(* IEC 61131-3 sources: plcassist-cli/packages/volt-lsp-iec/test-corpus/pro2193/Device/Plc Logic/Application/02 Processes/21 SER/2120 - Transfer Control/Products, 8 files *)

(* ---- TransferProducts_ChainToReject_WithCarrierPlatesFB.fb ---- *)
{attribute 'symbol' := 'none'}
{attribute 'monitoring_display' := 'ActState'}
FUNCTION_BLOCK TransferProducts_ChainToReject_WithCarrierPlatesFB
EXTENDS Transfer_BaseFB
IMPLEMENTS IModuleTransferExecute
VAR_INPUT
	chain					: IChain_WithCarrierPlates_TransferOuttake_Commands;
	reject					: IRejectStation_Base_Commands;
END_VAR
VAR
	gettingProduct			: ARRAY[1..GVL_Constants.ChainProductsForReject] OF BOOL;

	ActState :
	(
		StateNone							:= 0,
		StateRejectMovesInPosition			:= 100,
		StateRejectGetsProducts				:= 200,
		StateOpenProductCarriers			:= 250,
		StateCopyProductData				:= 300,
		StateFreeReject						:= 400,
		StateFinal							:= 999
	) DINT;

END_VAR

SUPER^();

// Enable manual control of Reject cylinders when chain is in safe position.
reject.ExternalManualControlEnabled := chain.InExactPosition();

END_FUNCTION_BLOCK

METHOD PUBLIC CheckIfTransferIsNeeded : BOOL
VAR_INPUT
	iParameter			: INT := 1;	// 0: Invalid, 1: Takeover Pos 1, etc.
END_VAR
VAR_INST
	product				: REFERENCE TO ProductType;
	i, j				: USINT;
END_VAR
// Go from first Reject vacuum, to the last.
FOR i := 1 TO GVL_Constants.ChainProductsForReject DO

	gettingProduct[i]		:= FALSE;

	// Copy reference to products from the chain
	product REF= chain.ReturnProduct(PersistentVars.RecipeVars.chainPos_Reject[i]);

	IF NOT __ISVALIDREF(product) THEN
		CONTINUE;
	END_IF

	FOR j := 1 TO GVL_Constants.MaxRejectReasonsTotal DO
		gettingProduct[i]	S= product.RejectReason[j] AND NOT product.RejectReasonIgnored[j];
	END_FOR

	gettingProduct[i]		S= product.UncountedReject;
	gettingProduct[i]		S= product.SampleShot;

	// When reject is after z unit, always reject all products
	IF NOT gettingProduct[i] AND NOT chain.ZUnitIsAfterReject THEN
		product.UncountedReject	:= TRUE;
		gettingProduct[i]	:= TRUE;
	END_IF

	CheckIfTransferIsNeeded	S= gettingProduct[i];
END_FOR
END_METHOD

METHOD PROTECTED Cyclic
State(actState	:= ActState);
END_METHOD

// Command to reset the module (Statemachine to zero state) in case of E-Stop
METHOD PUBLIC EStop : BOOL	// Returns true when drives are in standstill
CommandLock.ForceRelease();

ActState	:= StateNone;
EStop		:= TRUE;
END_METHOD

// Start transfer of products or labels between 2 units
METHOD PUBLIC ExecuteTransfer : BOOL
VAR_INPUT
	iParameter : INT := 1;	// 0: Invalid, 1: Takeover Pos 1, etc.
END_VAR
IF NOT CommandLock.Request(__POUNAME()) THEN
	RETURN;
END_IF

IF CommandLock.FirstCall THEN
	;
END_IF

takeoverPosition := iParameter;	// Copy parameters

IF ActState = StateNone THEN
	ActState := StateRejectMovesInPosition;
END_IF

IF ActState = StateFinal THEN
	ExecuteTransfer := CommandLock.Release(__POUNAME());
END_IF
END_METHOD

METHOD PROTECTED Execute_Sequence1
VAR_INST
	data				: WORD;
	product				: REFERENCE TO ProductType;
	result				: ARRAY[1..2] OF BOOL;
END_VAR
VAR
	i					: USINT;
END_VAR
CASE ActState OF
	StateNone:
		;

	StateRejectMovesInPosition:
		IF chain.InPosition(10.0) THEN
			ActState := StateRejectGetsProducts;
		END_IF

	StateRejectGetsProducts:

		IF State.Changed THEN
			Arrays.Bool_Reset(result);
			data := 0;
			FOR i := 1 TO GVL_Constants.ChainProductsForReject DO
				BitLogic.Load(data, gettingProduct[i], i);	// set a bit number when we transfer a product.
			END_FOR
		END_IF

		result[1]	:= result[1] OR_ELSE reject.GetProducts(data);

		IF chain.InExactPosition() THEN
			ActState := StateOpenProductCarriers;
		END_IF

	StateOpenProductCarriers:
		result[1]	:= result[1] OR_ELSE reject.GetProducts(data);
		result[2]	:= result[2] OR_ELSE chain.RejectOpenProductCarriers();

		IF Arrays.Bool_All(result, TRUE) THEN
			ActState := StateCopyProductData;
		END_IF

	StateCopyProductData:
		FOR i := 1 TO GVL_Constants.ChainProductsForReject DO

			IF NOT gettingProduct[i] THEN
				CONTINUE;
			END_IF

			// Copy reference to products from the chain
			product REF= chain.ReturnProduct(PersistentVars.RecipeVars.chainPos_Reject[i]);

			// Reject is not able to fail to transfer the product (like the Z Unit)
			reject.CopyProductStatus(i, product);
			chain.ClearProductCarrier(PersistentVars.RecipeVars.chainPos_Reject[i]);
			gettingProduct[i] := FALSE;

		END_FOR

		ActState := StateFreeReject;

	StateFreeReject:
		IF State.Changed THEN
			Arrays.Bool_Reset(result);
		END_IF

		// The last step of the product transfer must always be: TransferComplete()
		// This lets the Z Unit know that the transfer is done.
		// The Z Unit decides if it moves to the next Takeover position, or stack the products.
		result[1]	:= result[1] OR_ELSE reject.TransferComplete();
		result[2]	:= result[2] OR_ELSE chain.RejectCloseProductCarriers();

		IF Arrays.Bool_All(result, TRUE) THEN
			ActState := StateFinal;
		END_IF

	StateFinal:
		ActState := StateNone;
END_CASE
END_METHOD

// Command to stop a module (Statemachine to zero state)
METHOD PUBLIC Stop : BOOL	// Returns true when drives are in standstill
CommandLock.ForceRelease();

ActState	:= StateNone;
Stop		:= TRUE;
END_METHOD

// Transfer has started and is doing something
{attribute 'monitoring':='call'}
PROPERTY TransferBusy : BOOL
GET
VAR
END_VAR
TransferBusy	:= ActState <> StateNone;
END_GET
END_PROPERTY

(* ---- TransferProducts_ChainToRejectFB.fb ---- *)
{attribute 'symbol' := 'none'}
{attribute 'monitoring_display' := 'ActState'}
FUNCTION_BLOCK TransferProducts_ChainToRejectFB
EXTENDS Transfer_BaseFB
IMPLEMENTS IModuleTransferExecute
VAR_INPUT
	chain					: IChain_Base_TransferOuttake_Commands;
	reject					: IRejectStation_Base_Commands;
END_VAR
VAR
	gettingProduct			: ARRAY[1..GVL_Constants.ChainProductsForReject] OF BOOL;

	ActState :
	(
		StateNone							:= 0,
		StateRejectMovesInPosition			:= 100,
		StateRejectGetsProducts				:= 200,
		StateCopyProductData				:= 300,
		StateFreeReject						:= 400,
		StateFinal							:= 999
	) DINT;

END_VAR

SUPER^();

// Enable manual control of Reject cylinders when chain is in safe position.
reject.ExternalManualControlEnabled := chain.InExactPosition();

END_FUNCTION_BLOCK

METHOD PUBLIC CheckIfTransferIsNeeded : BOOL
VAR_INPUT
	iParameter			: INT := 1;	// 0: Invalid, 1: Takeover Pos 1, etc.
END_VAR
VAR_INST
	product				: REFERENCE TO ProductType;
	i, j				: USINT;
END_VAR
// Go from first Reject vacuum, to the last.
FOR i := 1 TO GVL_Constants.ChainProductsForReject DO

	gettingProduct[i]		:= FALSE;

	// Copy reference to products from the chain
	product REF= chain.ReturnProduct(PersistentVars.RecipeVars.chainPos_Reject[i]);

	IF NOT __ISVALIDREF(product) THEN
		EXIT;
	END_IF

	gettingProduct[i]		:= FALSE;

	FOR j := 1 TO GVL_Constants.MaxRejectReasonsTotal DO
		gettingProduct[i]	S= product.RejectReason[j] AND NOT product.RejectReasonIgnored[j];
	END_FOR

	gettingProduct[i]		S= product.UncountedReject;
	gettingProduct[i]		S= product.SampleShot;

	CheckIfTransferIsNeeded	S= gettingProduct[i];

	IF NOT gettingProduct[i] THEN
		EXIT;
	END_IF

END_FOR
END_METHOD

METHOD PROTECTED Cyclic
State(actState	:= ActState);
END_METHOD

// Command to reset the module (Statemachine to zero state) in case of E-Stop
METHOD PUBLIC EStop : BOOL	// Returns true when drives are in standstill
CommandLock.ForceRelease();

ActState	:= StateNone;
EStop		:= TRUE;
END_METHOD

// Start transfer of products or labels between 2 units
METHOD PUBLIC ExecuteTransfer : BOOL
VAR_INPUT
	iParameter : INT := 1;	// 0: Invalid, 1: Takeover Pos 1, etc.
END_VAR
IF NOT CommandLock.Request(__POUNAME()) THEN
	RETURN;
END_IF

IF CommandLock.FirstCall THEN
	;
END_IF

takeoverPosition := iParameter;	// Copy parameters

IF ActState = StateNone THEN
	ActState := StateRejectMovesInPosition;
END_IF

IF ActState = StateFinal THEN
	ExecuteTransfer := CommandLock.Release(__POUNAME());
END_IF
END_METHOD

METHOD PROTECTED Execute_Sequence1
VAR_INST
	data				: WORD;
	product				: REFERENCE TO ProductType;
	result				: ARRAY[1..2] OF BOOL;
END_VAR
VAR
	i					: USINT;
END_VAR
CASE ActState OF
	StateNone:
		;

	StateRejectMovesInPosition:
		IF chain.InExactPosition() THEN
			ActState := StateRejectGetsProducts;
		END_IF

	StateRejectGetsProducts:
		IF State.Changed THEN
			Arrays.Bool_Reset(result);
			data := 0;
			FOR i := 1 TO GVL_Constants.ChainProductsForReject DO
				BitLogic.Load(data, gettingProduct[i], i);	// set a bit number when we transfer a product.
			END_FOR
		END_IF

		result[1]	:= result[1] OR_ELSE reject.GetProducts(data);
		result[2]	:= TRUE;

		IF Arrays.Bool_All(result, TRUE) THEN
			ActState := StateCopyProductData;
		END_IF

	StateCopyProductData:
		FOR i := 1 TO GVL_Constants.ChainProductsForReject DO

			IF NOT gettingProduct[i] THEN
				CONTINUE;
			END_IF

			// Copy reference to products from the chain
			product REF= chain.ReturnProduct(PersistentVars.RecipeVars.chainPos_Reject[i]);

			// Reject is not able to fail to transfer the product (like the Z Unit)
			reject.CopyProductStatus(i, product);
			chain.ClearProductCarrier(PersistentVars.RecipeVars.chainPos_Reject[i]);
			gettingProduct[i] := FALSE;

		END_FOR

		ActState := StateFreeReject;

	StateFreeReject:
		IF State.Changed THEN
			Arrays.Bool_Reset(result);
		END_IF

		// The last step of the product transfer must always be: TransferComplete()
		// This lets the Z Unit know that the transfer is done.
		// The Z Unit decides if it moves to the next Takeover position, or stack the products.
		result[1]	:= result[1] OR_ELSE reject.TransferComplete();
		result[2]	:= TRUE;

		IF Arrays.Bool_All(result, TRUE) THEN
			ActState := StateFinal;
		END_IF

	StateFinal:
		ActState := StateNone;
END_CASE
END_METHOD

// Command to stop a module (Statemachine to zero state)
METHOD PUBLIC Stop : BOOL	// Returns true when drives are in standstill
CommandLock.ForceRelease();

ActState	:= StateNone;
Stop		:= TRUE;
END_METHOD

// Transfer has started and is doing something
{attribute 'monitoring':='call'}
PROPERTY TransferBusy : BOOL
GET
VAR
END_VAR
TransferBusy	:= ActState <> StateNone;
END_GET
END_PROPERTY

(* ---- TransferProducts_ChainToZ_WithCarrierPlatesFB.fb ---- *)
{attribute 'symbol' := 'none'}
{attribute 'monitoring_display' := 'ActState'}
FUNCTION_BLOCK TransferProducts_ChainToZ_WithCarrierPlatesFB
EXTENDS Transfer_BaseFB
IMPLEMENTS IModuleTransferExecute
VAR_INPUT
	chain					: IChain_WithCarrierPlates_TransferOuttake_Commands;
	zUnit					: IZUnit_ForChainWithServoRotate_Transfer_Commands;
END_VAR
VAR
	result					: ARRAY[1..2] OF BOOL;
	gettingProduct			: ARRAY[1..GVL_Constants.ChainProductsForZUnit] OF BOOL;

	ActState :
	(
		StateNone							:= 0,
		StateZUnitMovesInPosition			:= 100,
		StateZUnitGetsProducts				:= 200,
		StateZUnitOpenProductCarriers		:= 300,
		StateZUnitRetractWithProducts		:= 400,
		StateCopyProductData				:= 500,
		StateFreeZUnit						:= 600,
		StateFinal							:= 999
	) DINT;

END_VAR

SUPER^();

// Enable manual control of Z Unit motor when chain is in safe position.
zUnit.ExternalManualControlEnabled := TRUE; //chain.InExactPosition();

END_FUNCTION_BLOCK

METHOD PUBLIC CheckIfTransferIsNeeded : BOOL
VAR_INPUT
	iParameter			: INT := 1;	// 0: Invalid, 1: Takeover Pos 1, etc.
END_VAR
VAR_INST
	product				: REFERENCE TO ProductType;
	zUnitGripperFilled	: BOOL;
	data				: WORD;
END_VAR
VAR
	zUnithasProducts	: ARRAY[1..GVL_Constants.ChainProductsForZUnit] OF BOOL;
	i, j				: USINT;
END_VAR
zUnithasProducts	:= zUnit.HasProductForTransfer;

// Go from first Z Unit vacuum, to the last. First Z Unit vacuum is the last product on the chain.
FOR i := 1 TO GVL_Constants.ChainProductsForZUnit DO

	gettingProduct[i]		:= FALSE;

	// Copy reference to products from the chain
	data	:= PersistentVars.RecipeVars.chainPos_ZUnit[i] + chain.SelectedZUnitPosition - 1;
	product REF= chain.ReturnProduct(data);
//	product REF= chain.ReturnProduct(PersistentVars.RecipeVars.chainPos_ZUnit[i]);
//	product REF= chain.ReturnProduct(PersistentVars.RecipeVars.chainPos_ZUnit[i] + chain.SelectedZUnitPosition - 1);

	IF NOT __ISVALIDREF(product) THEN
		CONTINUE;
	END_IF

	// Check state of Z Unit gripper. Must be filled with products, up until this current one.
	zUnitGripperFilled		:= TRUE;
	IF i > 1 THEN
		FOR j := 1 TO i - 1 DO
			IF  NOT zUnithasProducts[j]
			AND NOT gettingProduct[j]
			THEN
				zUnitGripperFilled := FALSE;
				EXIT;
			END_IF
		END_FOR
	END_IF

	IF NOT zUnitGripperFilled THEN
		EXIT;
	END_IF

	IF (NOT product.UncountedReject OR chain.ZUnitIsAfterReject)	// Also get uncounted rejected products when the Z Unit is after the reject station.
	AND NOT product.SampleShot
	AND NOT zUnithasProducts[i]
	THEN
		gettingProduct[i]		:= TRUE;
		FOR j := 1 TO GVL_Constants.MaxRejectReasonsTotal DO
			gettingProduct[i]	R= product.RejectReason[j] AND NOT product.RejectReasonIgnored[j];
		END_FOR
	END_IF

	CheckIfTransferIsNeeded		S= gettingProduct[i];
END_FOR
END_METHOD

METHOD PROTECTED Cyclic
State(actState	:= ActState);
END_METHOD

// Command to reset the module (Statemachine to zero state) in case of E-Stop
METHOD PUBLIC EStop : BOOL	// Returns true when drives are in standstill
CommandLock.ForceRelease();

ActState	:= StateNone;
EStop		:= TRUE;
END_METHOD

// Start transfer of products or labels between 2 units
METHOD PUBLIC ExecuteTransfer : BOOL
VAR_INPUT
	iParameter : INT := 1;	// 0: Invalid, 1: Takeover Pos 1, etc.
END_VAR
IF NOT CommandLock.Request(__POUNAME()) THEN
	RETURN;
END_IF

IF CommandLock.FirstCall THEN
	;
END_IF

takeoverPosition := iParameter;	// Copy parameters

IF ActState = StateNone THEN
	ActState := StateZUnitMovesInPosition;
END_IF

IF ActState = StateFinal THEN
	ExecuteTransfer := CommandLock.Release(__POUNAME());
END_IF
END_METHOD

METHOD PROTECTED Execute_Sequence1
VAR_INST
	data				: WORD;
	shiftBits			: USINT;
	product				: REFERENCE TO ProductType;
	zUnithasProducts	: ARRAY[1..GVL_Constants.ChainProductsForZUnit] OF BOOL;
	result				: ARRAY[1..2] OF BOOL;
	Timer				: BTON;
END_VAR
VAR
	i					: USINT;
END_VAR
CASE ActState OF
	StateNone:
		;

	StateZUnitMovesInPosition:
		IF  zUnit.MoveToTakeover(chain.SelectedZUnitPosition)
		AND zUnit.ReadyForTransfer
		AND chain.InPosition(10.0)
		THEN
			ActState := StateZUnitGetsProducts;
		END_IF

	StateZUnitGetsProducts:
		IF State.Changed THEN
			Arrays.Bool_Reset(result);
			data				:= 0;
			FOR i := 1 TO GVL_Constants.ChainProductsForZUnit DO
				BitLogic.Load(data, gettingProduct[i], i);	// set a bit number for every product we transfer.
			END_FOR
		END_IF

		result[1]	:= result[1] OR_ELSE zUnit.GetProducts(data);		// var data can be changed by GetProducts!

		IF result[1] AND chain.InExactPosition() THEN
			Arrays.Bool_Reset(result);
			ActState := StateZUnitOpenProductCarriers;
		END_IF

	StateZUnitOpenProductCarriers:
		// Use SHL here to shift where on the chain to open the product carriers!
		// Because we have more product carriers than z axis vacuums
		// ZOpenProductCarrier 1 is at the bottom
		// ZOpenProductCarrier 3 matches with extend 1 on the Z axis
		CASE chain.SelectedZUnitPosition OF
			1:	shiftBits	:= 3;
			2:	shiftBits	:= 2;
			3:	shiftBits	:= 1;
			4:	shiftBits	:= 0;
		END_CASE

		IF chain.ZOpenProductCarriers(SHL(data, shiftBits)) THEN
			ActState := StateZUnitRetractWithProducts;
		END_IF

	StateZUnitRetractWithProducts:
		IF state.Changed THEN
			Timer.Reset();
		END_IF

		IF Timer.Set(In := TRUE, Pt := 0.2) THEN
			chain.ZCloseProductCarriers();
		END_IF

		IF zUnit.RetractWithProducts() THEN
			ActState := StateCopyProductData;
		END_IF

	StateCopyProductData:
		zUnithasProducts := zUnit.HasProductForTransfer;

		FOR i := 1 TO GVL_Constants.ChainProductsForZUnit DO

			IF NOT gettingProduct[i] THEN
				CONTINUE;
			END_IF

			// Copy reference to products from the chain
			data	:= PersistentVars.RecipeVars.chainPos_ZUnit[i] + chain.SelectedZUnitPosition - 1;
			product REF= chain.ReturnProduct(data);
//			product REF= chain.ReturnProduct(PersistentVars.RecipeVars.chainPos_ZUnit[i]);

			IF NOT __ISVALIDREF(product) THEN
				LogPlc.Error('Product was lost on the chain. This should not happen ???!?');
			ELSIF NOT zUnithasProducts[i] THEN		// Failed to transfer product?

				IF chain.ZUnitIsAfterReject THEN
					product.Present			:= FALSE;	// Assume product is missing. Cycle will stop when sensor detects a product after Z unit.
				ELSE
					product.UncountedReject	:= TRUE;	// The reject station can remove the product from the chain.
				END_IF

			ELSE
				zUnit.CopyProductStatus(1, i, product);
				chain.ClearProductCarrier(data);
	//			chain.ClearProductCarrier(PersistentVars.RecipeVars.chainPos_ZUnit[i]);
			END_IF
			gettingProduct[i] := FALSE;
		END_FOR

		IF Arrays.Bool_All(zUnithasProducts, TRUE) THEN		// Only increment when Z Unit has a full gripper
			chain.IncrementActiveOrderSelect();
		END_IF

		Arrays.Bool_Reset(result);

		ActState := StateFreeZUnit;

	StateFreeZUnit:
		// The last step of the product transfer must always be: TransferComplete()
		// This lets the Z Unit know that the transfer is done.
		// The Z Unit decides if it moves to the next Takeover position, or stack the products.
		result[1]	:= result[1] OR_ELSE zUnit.TransferComplete(chain.SelectedZUnitPosition);
		result[2]	:= result[2] OR_ELSE chain.ZCloseProductCarriers();

		IF Arrays.Bool_All(result, TRUE) THEN
			ActState := StateFinal;
		END_IF

	StateFinal:
		ActState := StateNone;
END_CASE
END_METHOD

// Command to stop a module (Statemachine to zero state)
METHOD PUBLIC Stop : BOOL	// Returns true when drives are in standstill
CommandLock.ForceRelease();

ActState	:= StateNone;
Stop		:= TRUE;
END_METHOD

// Transfer has started and is doing something
{attribute 'monitoring':='call'}
PROPERTY TransferBusy : BOOL
GET
VAR
END_VAR
TransferBusy	:= ActState <> StateNone;
END_GET
END_PROPERTY

(* ---- TransferProducts_ChainToZFB.fb ---- *)
{attribute 'symbol' := 'none'}
{attribute 'monitoring_display' := 'ActState'}
FUNCTION_BLOCK TransferProducts_ChainToZFB
EXTENDS Transfer_BaseFB
IMPLEMENTS IModuleTransferExecute
VAR_INPUT
	chain					: IChain_Base_TransferOuttake_Commands;
	zUnit					: IZUnit_ForChainWithServoRotate_Transfer_Commands;
END_VAR
VAR
	result					: ARRAY[1..2] OF BOOL;
	gettingProduct			: ARRAY[1..GVL_Constants.ChainProductsForZUnit] OF BOOL;

	ActState :
	(
		StateNone							:= 0,
		StateZUnitMovesInPosition			:= 100,
		StateZUnitGetsProducts				:= 200,
		StateCopyProductData				:= 300,
		StateFreeZUnit						:= 400,
		StateFinal							:= 999
	) DINT;

END_VAR

SUPER^();

// Enable manual control of Z Unit motor when chain is in safe position.
zUnit.ExternalManualControlEnabled := TRUE; //chain.InExactPosition();

END_FUNCTION_BLOCK

METHOD PUBLIC CheckIfTransferIsNeeded : BOOL
VAR_INPUT
	iParameter			: INT := 1;	// 0: Invalid, 1: Takeover Pos 1, etc.
END_VAR
VAR_INST
	product				: REFERENCE TO ProductType;
	zUnitGripperFilled	: BOOL;
END_VAR
VAR
	zUnithasProducts	: ARRAY[1..GVL_Constants.ChainProductsForZUnit] OF BOOL;
	i, j				: USINT;
END_VAR
zUnithasProducts	:= zUnit.HasProductForTransfer;

// Go from first Z Unit vacuum, to the last. First Z Unit vacuum is the last product on the chain.
FOR i := 1 TO GVL_Constants.ChainProductsForZUnit DO

	// Copy reference to products from the chain
	product REF= chain.ReturnProduct(PersistentVars.RecipeVars.chainPos_ZUnit[i]);

	IF NOT __ISVALIDREF(product) THEN
		CONTINUE;
	END_IF

	// Check state of Z Unit gripper. Must be filled with products, up until this current one.
	zUnitGripperFilled	:= TRUE;
	IF i > 1 THEN
		FOR j := 1 TO i - 1 DO
			IF  NOT zUnithasProducts[j]
			AND NOT gettingProduct[j]
			THEN
				zUnitGripperFilled := FALSE;
				EXIT;
			END_IF
		END_FOR
	END_IF

	IF NOT zUnitGripperFilled THEN
		EXIT;
	END_IF

	IF (NOT product.UncountedReject OR chain.ZUnitIsAfterReject)	// Also get uncounted rejected products when the Z Unit is after the reject station.
	AND NOT product.SampleShot
	AND NOT zUnithasProducts[i]
	THEN
		gettingProduct[i]		:= TRUE;
		FOR j := 1 TO GVL_Constants.MaxRejectReasonsTotal DO
			gettingProduct[i]	R= product.RejectReason[j] AND NOT product.RejectReasonIgnored[j];
		END_FOR
	ELSE
		gettingProduct[i]		:= FALSE;
	END_IF

	CheckIfTransferIsNeeded		S= gettingProduct[i];

	IF NOT gettingProduct[i] THEN
		EXIT;
	END_IF

END_FOR
END_METHOD

METHOD PROTECTED Cyclic
State(actState	:= ActState);
END_METHOD

// Command to reset the module (Statemachine to zero state) in case of E-Stop
METHOD PUBLIC EStop : BOOL	// Returns true when drives are in standstill
CommandLock.ForceRelease();

ActState	:= StateNone;
EStop		:= TRUE;
END_METHOD

// Start transfer of products or labels between 2 units
METHOD PUBLIC ExecuteTransfer : BOOL
VAR_INPUT
	iParameter : INT := 1;	// 0: Invalid, 1: Takeover Pos 1, etc.
END_VAR
IF NOT CommandLock.Request(__POUNAME()) THEN
	RETURN;
END_IF

IF CommandLock.FirstCall THEN
	;
END_IF

takeoverPosition := iParameter;	// Copy parameters

IF ActState = StateNone THEN
	ActState := StateZUnitMovesInPosition;
END_IF

IF ActState = StateFinal THEN
	ExecuteTransfer := CommandLock.Release(__POUNAME());
END_IF
END_METHOD

METHOD PROTECTED Execute_Sequence1
VAR_INST
	data				: WORD;
	product				: REFERENCE TO ProductType;
	zUnithasProducts	: ARRAY[1..GVL_Constants.ChainProductsForZUnit] OF BOOL;
END_VAR
VAR
	i					: USINT;
END_VAR
CASE ActState OF
	StateNone:
		;

	StateZUnitMovesInPosition:
		IF  zUnit.MoveToTakeover(1)
		AND zUnit.ReadyForTransfer
		AND chain.InExactPosition()
		THEN
			ActState := StateZUnitGetsProducts;
		END_IF

	StateZUnitGetsProducts:
		IF State.Changed THEN
			Arrays.Bool_Reset(result);
			data := 0;
			FOR i := 1 TO GVL_Constants.ChainProductsForZUnit DO
				BitLogic.Load(data, gettingProduct[i], i);	// set a bit number for every product we transfer.
			END_FOR
		END_IF

		IF result[1] := zUnit.GetProducts(data) THEN
			ActState := StateCopyProductData;
		END_IF

	StateCopyProductData:
		zUnithasProducts := zUnit.HasProductForTransfer;

		FOR i := 1 TO GVL_Constants.ChainProductsForZUnit DO

			IF NOT gettingProduct[i] THEN
				CONTINUE;
			END_IF

			// Copy reference to products from the chain
			product REF= chain.ReturnProduct(PersistentVars.RecipeVars.chainPos_ZUnit[i]);

			IF NOT __ISVALIDREF(product) THEN
				LogPlc.Error('Product was lost on the chain. This should not happen ???!?');
			ELSIF NOT zUnithasProducts[i] THEN		// Failed to transfer product?

				IF chain.ZUnitIsAfterReject THEN
					product.Present			:= FALSE;	// Assume product is missing. Cycle will stop when sensor detects a product after Z unit.
				ELSE
					product.UncountedReject	:= TRUE;	// The reject station can remove the product from the chain.
				END_IF

			ELSE
				zUnit.CopyProductStatus(1, i, product);
				chain.ClearProductCarrier(PersistentVars.RecipeVars.chainPos_ZUnit[i]);
			END_IF
			gettingProduct[i] := FALSE;
		END_FOR

		ActState := StateFreeZUnit;

	StateFreeZUnit:
		IF State.Changed THEN
			Arrays.Bool_Reset(result);
		END_IF

		// The last step of the product transfer must always be: TransferComplete()
		// This lets the Z Unit know that the transfer is done.
		// The Z Unit decides if it moves to the next Takeover position, or stack the products.
		result[1]	:= result[1] OR_ELSE zUnit.TransferComplete();
		result[2]	:= TRUE;

		IF Arrays.Bool_All(result, TRUE) THEN
			ActState := StateFinal;
		END_IF

	StateFinal:
		ActState := StateNone;
END_CASE
END_METHOD

// Command to stop a module (Statemachine to zero state)
METHOD PUBLIC Stop : BOOL	// Returns true when drives are in standstill
CommandLock.ForceRelease();

ActState	:= StateNone;
Stop		:= TRUE;
END_METHOD

// Transfer has started and is doing something
{attribute 'monitoring':='call'}
PROPERTY TransferBusy : BOOL
GET
VAR
END_VAR
TransferBusy	:= ActState <> StateNone;
END_GET
END_PROPERTY

(* ---- TransferProducts_XuToChain_WithCarrierPlatesFB.fb ---- *)
{attribute 'symbol' := 'none'}
{attribute 'monitoring_display' := 'ActState'}
FUNCTION_BLOCK TransferProducts_XuToChain_WithCarrierPlatesFB
EXTENDS Transfer_BaseFB
IMPLEMENTS IModuleTransferExecuteWithPrepare
VAR_INPUT
	xuUnit					: IXuUnit_ForChain_Transfer_Commands;
	chain					: IChain_WithCarrierPlates_TransferIntake_Commands;
END_VAR
VAR
	ActState :
	(
		StateNone							:= 0,
		StatePrepareTransfer				:= 50,
		StateCheckPayload					:= 100,
		StateXuUnitMovesToHalfwayTakeover	:= 200,
		StateXuUnitMovesToTakeover			:= 300,
		StateXuUnitReleasesProducts			:= 400,
		StateXuUnitMovesToParking			:= 500,
		StateFreeChain						:= 600,
		StateFinal							:= 999
	) DINT;

END_VAR

SUPER^();

END_FUNCTION_BLOCK

// Check if a transfer is needed
METHOD PUBLIC CheckIfTransferIsNeeded : BOOL
VAR_INPUT
	iParameter			: INT := 1;	// 0: Invalid, 1: Takeover Pos 1, etc.
END_VAR
VAR_INST
	xuUnitVacuum		: WORD;
	product				: ProductType;
END_VAR
// Xu unit has vacuum high that is needed for this Takeover position
xuUnitVacuum	:= 0;
CASE iParameter OF
	1:	xuUnitVacuum.Vacuum01	:= TRUE;
	2:	xuUnitVacuum.Vacuum02	:= TRUE;
	3:	xuUnitVacuum.Vacuum03	:= TRUE;
END_CASE

CheckIfTransferIsNeeded	S= xuUnit.HasVacuumHigh(xuUnitVacuum);

// Xu unit has at least 1 product in the gripper. We need a transfer.
//CheckIfTransferIsNeeded	S= xuUnit.HasPayload <> enumPayload.None;

// Running in semi-auto mode without setting vacuums.
CheckIfTransferIsNeeded	S= SER.OperationMode = SER_OperationModeType.SemiAuto AND HMI.SemiAutoMode = enumSemiAutoModeType.WithoutVacuums;

CASE iParameter OF
	1:
		product					:= xuUnit.ProductData_Get(product := 10);
		CheckIfTransferIsNeeded	R= product.ToShute;
		product					:= xuUnit.ProductData_Get(product := 7);
		CheckIfTransferIsNeeded	R= product.ToShute;
		product					:= xuUnit.ProductData_Get(product := 4);
		CheckIfTransferIsNeeded	R= product.ToShute;
		product					:= xuUnit.ProductData_Get(product := 1);
		CheckIfTransferIsNeeded	R= product.ToShute;
	2:
		product					:= xuUnit.ProductData_Get(product := 11);
		CheckIfTransferIsNeeded	R= product.ToShute;
		product					:= xuUnit.ProductData_Get(product := 8);
		CheckIfTransferIsNeeded	R= product.ToShute;
		product					:= xuUnit.ProductData_Get(product := 5);
		CheckIfTransferIsNeeded	R= product.ToShute;
		product					:= xuUnit.ProductData_Get(product := 2);
		CheckIfTransferIsNeeded	R= product.ToShute;
	3:
		product					:= xuUnit.ProductData_Get(product := 12);
		CheckIfTransferIsNeeded	R= product.ToShute;
		product					:= xuUnit.ProductData_Get(product := 9);
		CheckIfTransferIsNeeded	R= product.ToShute;
		product					:= xuUnit.ProductData_Get(product := 6);
		CheckIfTransferIsNeeded	R= product.ToShute;
		product					:= xuUnit.ProductData_Get(product := 3);
		CheckIfTransferIsNeeded	R= product.ToShute;
END_CASE
END_METHOD

METHOD PROTECTED Cyclic
State(actState	:= ActState);
END_METHOD

// Command to reset the module (Statemachine to zero state) in case of E-Stop
METHOD PUBLIC EStop : BOOL	// Returns true when drives are in standstill
CommandLock.ForceRelease();

ActState	:= StateNone;
EStop		:= TRUE;
END_METHOD

// Start transfer of products or labels between 2 units
METHOD PUBLIC ExecuteTransfer : BOOL
VAR_INPUT
	iParameter : INT := 1;	// 0: Invalid, 1: Takeover Pos 1, etc.
END_VAR
IF NOT CommandLock.Request(__POUNAME()) THEN
	RETURN;
END_IF

IF CommandLock.FirstCall THEN
	;
END_IF

takeoverPosition	:= iParameter;	// Copy parameters

IF ActState = StateNone OR ActState = StatePrepareTransfer THEN
	ActState := StateCheckPayload;
END_IF

IF ActState = StateFinal THEN
	ExecuteTransfer := CommandLock.Release(__POUNAME());
END_IF
END_METHOD

METHOD PROTECTED Execute_Sequence1
VAR_INST
	xuUnitVacuum		: WORD;
	result				: ARRAY[1..2] OF BOOL;
	almostSafe			: BOOL;
END_VAR
CASE ActState OF
	StateNone:
		;

	StatePrepareTransfer:
		IF State.Changed THEN
			Arrays.Bool_Reset(result);
			xuUnitVacuum	:= 0;
			CASE takeoverPosition OF
				1:	xuUnitVacuum.Vacuum01	:= TRUE;
				2:	xuUnitVacuum.Vacuum02	:= TRUE;
				3:	xuUnitVacuum.Vacuum03	:= TRUE;
			END_CASE
			xuUnit.ForceReleaseLock();
		END_IF

		IF xuUnit.HasVacuumHigh(xuUnitVacuum)
		OR (SER.OperationMode = SER_OperationModeType.SemiAuto AND HMI.SemiAutoMode = enumSemiAutoModeType.WithoutVacuums)
		OR SER.ActState = PACK_ML.State.Starting
		THEN
			IF  chain.InPosition(10)
			AND chain.ProductsNeeded
			THEN
				result[1]	:= result[1] OR_ELSE xuUnit.MoveToInFrontOfChain();
			END_IF
			IF  chain.InExactPosition()
			AND chain.ProductsNeeded
			THEN
				result[2]	:= result[2] OR_ELSE chain.XuOpenProductCarriers();
			END_IF
		END_IF

	StateCheckPayload:
		// Check if all products are present on the Xu Unit gripper.
		// Or the cycle has just started, the first cycle it is allowed to transfer an incomplete gripper.
		IF State.Changed THEN
			xuUnitVacuum	:= 0;
			CASE takeoverPosition OF
				1:	xuUnitVacuum.Vacuum01	:= TRUE;
				2:	xuUnitVacuum.Vacuum02	:= TRUE;
				3:	xuUnitVacuum.Vacuum03	:= TRUE;
			END_CASE
		END_IF

		IF xuUnit.HasVacuumHigh(xuUnitVacuum)
//		IF xuUnit.HasPayload = enumPayload._All
		OR (SER.OperationMode = SER_OperationModeType.SemiAuto AND HMI.SemiAutoMode = enumSemiAutoModeType.WithoutVacuums)
		OR SER.ActState = PACK_ML.State.Starting
		THEN
			ActState := StateXuUnitMovesToHalfwayTakeover;
		END_IF

	StateXuUnitMovesToHalfwayTakeover:
		IF State.Changed THEN
			;//xuUnit.MoveToHalfway();
		END_IF

		IF  chain.InPosition(10)
		AND chain.ProductsNeeded
		THEN
			result[1]	:= result[1] OR_ELSE xuUnit.MoveToInFrontOfChain();
		END_IF

		IF  chain.InExactPosition()
		AND chain.ProductsNeeded
//		AND xuUnit.ShiftToTransfer()
		THEN
			IF chain.XuOpenProductCarriers() THEN
				ActState := StateXuUnitMovesToTakeover;
			END_IF
		END_IF

	StateXuUnitMovesToTakeover:
		IF xuUnit.MoveToTakeover(1) THEN
			ActState := StateXuUnitReleasesProducts;
		END_IF

	StateXuUnitReleasesProducts:
		IF State.Changed THEN
			Arrays.Bool_Reset(result);
			xuUnitVacuum	:= 0;
			CASE takeoverPosition OF
				1:

					chain.CopyProductStatus(productNo	:= 1,	product		:= xuUnit.ProductData_Get(product := 10,	clearLastProduct := TRUE, clearData := TRUE));
					chain.CopyProductStatus(productNo	:= 2,	product		:= xuUnit.ProductData_Get(product := 7,		clearLastProduct := TRUE, clearData := TRUE));
					chain.CopyProductStatus(productNo	:= 3,	product		:= xuUnit.ProductData_Get(product := 4,		clearLastProduct := TRUE, clearData := TRUE));
					chain.CopyProductStatus(productNo	:= 4,	product		:= xuUnit.ProductData_Get(product := 1,		clearLastProduct := TRUE, clearData := TRUE));
					xuUnitVacuum.Vacuum01	:= TRUE;

				2:
					chain.CopyProductStatus(productNo	:= 1,	product		:= xuUnit.ProductData_Get(product := 11,	clearLastProduct := TRUE, clearData := TRUE));
					chain.CopyProductStatus(productNo	:= 2,	product		:= xuUnit.ProductData_Get(product := 8,		clearLastProduct := TRUE, clearData := TRUE));
					chain.CopyProductStatus(productNo	:= 3,	product		:= xuUnit.ProductData_Get(product := 5,		clearLastProduct := TRUE, clearData := TRUE));
					chain.CopyProductStatus(productNo	:= 4,	product		:= xuUnit.ProductData_Get(product := 2,		clearLastProduct := TRUE, clearData := TRUE));
					xuUnitVacuum.Vacuum02	:= TRUE;
				3:
					chain.CopyProductStatus(productNo	:= 1,	product		:= xuUnit.ProductData_Get(product := 12,	clearLastProduct := FALSE, clearData := TRUE));
					chain.CopyProductStatus(productNo	:= 2,	product		:= xuUnit.ProductData_Get(product := 9,		clearLastProduct := FALSE, clearData := TRUE));
					chain.CopyProductStatus(productNo	:= 3,	product		:= xuUnit.ProductData_Get(product := 6,		clearLastProduct := FALSE, clearData := TRUE));
					chain.CopyProductStatus(productNo	:= 4,	product		:= xuUnit.ProductData_Get(product := 3,		clearLastProduct := FALSE, clearData := TRUE));
					xuUnitVacuum.Vacuum03	:= TRUE;
			END_CASE

(*			// Not possible for a direct copy of the status because the shift cylincer on the Xu shifts the products around.
			chain.CopyProductStatus(productNo	:= 1,	product		:= xuUnit.ProductData_Get(product := 1));
			chain.CopyProductStatus(productNo	:= 2,	product		:= xuUnit.ProductData_Get(product := 4));
			chain.CopyProductStatus(productNo	:= 3,	product		:= xuUnit.ProductData_Get(product := 2));
			chain.CopyProductStatus(productNo	:= 4,	product		:= xuUnit.ProductData_Get(product := 5));
			chain.CopyProductStatus(productNo	:= 5,	product		:= xuUnit.ProductData_Get(product := 3));
			chain.CopyProductStatus(productNo	:= 6,	product		:= xuUnit.ProductData_Get(product := 6));
*)
(*
			FOR i := 1 TO GVL_Constants.ChainProductsForXuUnit DO
				chain.CopyProductStatus(
					productNo	:= i,
					product		:= xuUnit.ProductData_Get(product := i));
			END_FOR
*)

		END_IF

		// Xu Unit releases all vacuums; returns true after a timeout.
		result[1]	:= result[1] OR_ELSE xuUnit.ReleaseProducts(xuUnitVacuum);
		result[2]	:= result[2] OR_ELSE chain.XuCloseProductCarriers();

		IF Arrays.Bool_All(result, TRUE) THEN
			ActState := StateXuUnitMovesToParking;
		END_IF

	StateXuUnitMovesToParking:
		IF State.Changed THEN
			Arrays.Bool_Reset(result);
		END_IF

		IF takeoverPosition = 3
		OR xuUnit.HasPayload = enumPayload.None
		THEN
			result[1]	:= result[1] OR_ELSE xuUnit.MoveToParking(almostSafe => almostSafe);
		ELSE
			result[1]	:= result[1] OR_ELSE xuUnit.MoveToHalfway();
		END_IF

		IF xuUnit.InSafePosForChain THEN
			ActState := StateFreeChain;
		END_IF

	StateFreeChain:
		// The last step of the product transfer must always be: TransferComplete()
		// This lets the Z Unit know that the transfer is done.
		// The Z Unit decides if it moves to the next Takeover position, or stack the products.
		IF takeoverPosition = 3
		OR xuUnit.HasPayload = enumPayload.None
		THEN
			result[1]	:= result[1] OR_ELSE xuUnit.MoveToParking(almostSafe => almostSafe);
		ELSE
			result[1]	:= result[1] OR_ELSE xuUnit.MoveToHalfway();
		END_IF

		result[2]	:= result[2] OR_ELSE chain.TransferComplete(takeoverPosition);
//		AND xuUnit.ShiftToTakeout()

		IF (result[1] OR almostSafe) AND result[2] THEN
			ActState := StateFinal;
		END_IF

	StateFinal:
		ActState := StateNone;
END_CASE
END_METHOD

// Prepare transfer of products while Y axis is still moving
METHOD PUBLIC PrepareTransfer : BOOL
VAR_INPUT
	iParameter : INT := 1;	// 0: Invalid, 1: Takeover Pos 1, etc.
END_VAR
IF NOT CommandLock.Request(__POUNAME()) THEN
	RETURN;
END_IF

takeoverPosition	:= iParameter;	// Copy parameters

IF ActState = StateNone THEN
	ActState := StatePrepareTransfer;
END_IF

PrepareTransfer := CommandLock.Release(__POUNAME());
END_METHOD

// Command to stop a module (Statemachine to zero state)
METHOD PUBLIC Stop : BOOL	// Returns true when drives are in standstill
CommandLock.ForceRelease();

ActState	:= StateNone;
Stop		:= TRUE;
END_METHOD

// Transfer has started and is doing something
{attribute 'monitoring':='call'}
PROPERTY TransferBusy : BOOL
GET
VAR
END_VAR
TransferBusy	:= ActState <> StateNone;
END_GET
END_PROPERTY

(* ---- TransferProducts_XuToChainFB.fb ---- *)
{attribute 'symbol' := 'none'}
{attribute 'monitoring_display' := 'ActState'}
FUNCTION_BLOCK TransferProducts_XuToChainFB
EXTENDS Transfer_BaseFB
IMPLEMENTS IModuleTransferExecute
VAR_INPUT
	xuUnit					: IXuUnit_ForChain_Transfer_Commands;
	chain					: IChain_Base_TransferIntake_Commands;
END_VAR
VAR
	ActState :
	(
		StateNone							:= 0,
		StateCheckPayload					:= 100,
		StateXuUnitMovesToHalfwayTakeover	:= 200,
		StateXuUnitMovesToTakeover			:= 300,
		StateXuUnitReleasesProducts			:= 400,
		StateXuUnitMovesToParking			:= 500,
		StateFreeChain						:= 600,
		StateFinal							:= 999
	) DINT;

END_VAR

SUPER^();

END_FUNCTION_BLOCK

// Check if a transfer is needed
METHOD PUBLIC CheckIfTransferIsNeeded : BOOL
VAR_INPUT
	iParameter			: INT := 1;	// 0: Invalid, 1: Takeover Pos 1, etc.
END_VAR
// Xu unit has at least 1 product in the gripper. We need a transfer.
CheckIfTransferIsNeeded	S= xuUnit.HasPayload <> enumPayload.None;

// Running in semi-auto mode without setting vacuums.
CheckIfTransferIsNeeded	S= SER.OperationMode = SER_OperationModeType.SemiAuto AND HMI.SemiAutoMode = enumSemiAutoModeType.WithoutVacuums;
END_METHOD

METHOD PROTECTED Cyclic
State(actState	:= ActState);
END_METHOD

// Command to reset the module (Statemachine to zero state) in case of E-Stop
METHOD PUBLIC EStop : BOOL	// Returns true when drives are in standstill
CommandLock.ForceRelease();

ActState	:= StateNone;
EStop		:= TRUE;
END_METHOD

// Start transfer of products or labels between 2 units
METHOD PUBLIC ExecuteTransfer : BOOL
VAR_INPUT
	iParameter : INT := 1;	// 0: Invalid, 1: Takeover Pos 1, etc.
END_VAR
IF NOT CommandLock.Request(__POUNAME()) THEN
	RETURN;
END_IF

IF CommandLock.FirstCall THEN
	;
END_IF

takeoverPosition := iParameter;	// Copy parameters

IF ActState = StateNone THEN
	ActState := StateCheckPayload;
END_IF

IF ActState = StateFinal THEN
	ExecuteTransfer := CommandLock.Release(__POUNAME());
END_IF
END_METHOD

METHOD PROTECTED Execute_Sequence1
VAR_INST
	result				: ARRAY[1..2] OF BOOL;
END_VAR
CASE ActState OF
	StateNone:
		;

	StateCheckPayload:
		// Check if all products are present on the Xu Unit gripper.
		// Or the cycle has just started, the first cycle it is allowed to transfer an incomplete gripper.
		IF xuUnit.HasPayload = enumPayload._All
		OR SER.OperationMode = SER_OperationModeType.SemiAuto
		OR SER.ActState = PACK_ML.State.Starting
		THEN
			ActState := StateXuUnitMovesToHalfwayTakeover;
		END_IF

	StateXuUnitMovesToHalfwayTakeover:
		IF State.Changed THEN
			xuUnit.MoveToHalfway();
		END_IF

		IF  chain.InExactPosition()
		AND chain.ProductsNeeded
//		AND xuUnit.ShiftToTransfer()
		THEN
			ActState := StateXuUnitMovesToTakeover;
		END_IF

	StateXuUnitMovesToTakeover:
		IF xuUnit.MoveToTakeover(1) THEN
			ActState := StateXuUnitReleasesProducts;
		END_IF

	StateXuUnitReleasesProducts:
		IF State.Changed THEN

			// Not possible for a direct copy of the status because the shift cylincer on the Xu shifts the products around.

			chain.CopyProductStatus(productNo	:= 1,	product		:= xuUnit.ProductData_Get(product := 1));
			chain.CopyProductStatus(productNo	:= 2,	product		:= xuUnit.ProductData_Get(product := 4));
			chain.CopyProductStatus(productNo	:= 3,	product		:= xuUnit.ProductData_Get(product := 2));
//			chain.CopyProductStatus(productNo	:= 4,	product		:= xuUnit.ProductData_Get(product := 5));
//			chain.CopyProductStatus(productNo	:= 5,	product		:= xuUnit.ProductData_Get(product := 3));
//			chain.CopyProductStatus(productNo	:= 6,	product		:= xuUnit.ProductData_Get(product := 6));

//			FOR i := 1 TO GVL_Constants.ChainProductsForXuUnit DO
//				chain.CopyProductStatus(
//					productNo	:= i,
//					product		:= xuUnit.ProductData_Get(product := i));
//			END_FOR

		END_IF

		// Xu Unit releases all vacuums; returns true after a timeout.
		IF xuUnit.ReleaseProducts(AllVacuums) THEN
			ActState := StateXuUnitMovesToParking;
		END_IF

	StateXuUnitMovesToParking:
		xuUnit.MoveToParking();

		IF xuUnit.InSafePosForChain THEN
			ActState := StateFreeChain;
		END_IF

	StateFreeChain:
		// The last step of the product transfer must always be: TransferComplete()
		// This lets the Z Unit know that the transfer is done.
		// The Z Unit decides if it moves to the next Takeover position, or stack the products.
		IF chain.TransferComplete(takeoverPosition)
//		AND xuUnit.ShiftToTakeout()
		AND xuUnit.MoveToParking()
		THEN
			ActState := StateFinal;
		END_IF

	StateFinal:
		ActState := StateNone;
END_CASE
END_METHOD

// Command to stop a module (Statemachine to zero state)
METHOD PUBLIC Stop : BOOL	// Returns true when drives are in standstill
CommandLock.ForceRelease();

ActState	:= StateNone;
Stop		:= TRUE;
END_METHOD

// Transfer has started and is doing something
{attribute 'monitoring':='call'}
PROPERTY TransferBusy : BOOL
GET
VAR
END_VAR
TransferBusy	:= ActState <> StateNone;
END_GET
END_PROPERTY

(* ---- TransferProducts_XuToShuteFB.fb ---- *)
{attribute 'symbol' := 'none'}
{attribute 'monitoring_display' := 'ActState'}
FUNCTION_BLOCK TransferProducts_XuToShuteFB
EXTENDS Transfer_BaseFB
IMPLEMENTS IModuleTransferExecute
VAR_INPUT
	xuUnit					: IXuUnit_Default_Transfer_Commands;
	conveyor				: IConveyor_Reject_Move_Commands;
	statistics				: IAddProductionStats;
	PulseOutput				: PulseActuatorFB;
END_VAR
VAR
	ActState :
	(
		StateNone							:= 0,
		StateXuUnitMovesToTakeover			:= 100,
		StateXuUnitReleasesProducts			:= 200,
		StateXuUnitMovesToParking			:= 300,
		StateFinal							:= 999
	) DINT;
END_VAR

SUPER^();

END_FUNCTION_BLOCK

// Check if a transfer is needed
METHOD PUBLIC CheckIfTransferIsNeeded : BOOL
VAR_INPUT
	iParameter			: INT := 1;	// 0: Invalid, 1: Takeover Pos 1, etc.
END_VAR
VAR_INST
	xuUnitVacuum	: WORD;
END_VAR
// Xu unit has vacuum high that is needed for this Takeover position
xuUnitVacuum	:= 0;
CASE iParameter OF
	1:	xuUnitVacuum.Vacuum01	:= TRUE;
	2:	xuUnitVacuum.Vacuum02	:= TRUE;
	3:	xuUnitVacuum.Vacuum03	:= TRUE;
END_CASE

CheckIfTransferIsNeeded	S= xuUnit.HasVacuumHigh(xuUnitVacuum);
END_METHOD

METHOD PROTECTED Cyclic
State(actState	:= ActState);

PulseOutput(
	pulseTimeLow	:= ,
	pulseTimeHigh	:= );
END_METHOD

// Command to reset the module (Statemachine to zero state) in case of E-Stop
METHOD PUBLIC EStop : BOOL	// Returns true when drives are in standstill
CommandLock.ForceRelease();

ActState	:= StateNone;
EStop		:= TRUE;
END_METHOD

// Start transfer of products or labels between 2 units
METHOD PUBLIC ExecuteTransfer : BOOL
VAR_INPUT
	iParameter : INT := 1;	// 0: Invalid, 1: Takeover Pos 1, etc.
END_VAR
IF NOT CommandLock.Request(__POUNAME()) THEN
	RETURN;
END_IF

IF CommandLock.FirstCall THEN
	;
END_IF

takeoverPosition := iParameter;	// Copy parameters

IF ActState = StateNone THEN
	ActState := StateXuUnitMovesToTakeover;
END_IF

IF ActState = StateFinal THEN
	ExecuteTransfer := CommandLock.Release(__POUNAME());
END_IF
END_METHOD

METHOD PROTECTED Execute_Sequence1
VAR_INST
	xuUnitVacuum		: WORD;
	result				: ARRAY[1..1] OF BOOL;
	almostSafe			: BOOL;
	product				: ProductType;
	Timer				: BTON;
END_VAR
CASE ActState OF
	StateNone:
		;

	StateXuUnitMovesToTakeover:
		IF xuUnit.MoveToTakeover(2) THEN
			ActState := StateXuUnitReleasesProducts;
		END_IF

	StateXuUnitReleasesProducts:
		IF statistics = 0 THEN
			RETURN;
		END_IF

		IF State.Changed THEN
			conveyor.MoveStep();
			Timer.Reset();
			Arrays.Bool_Reset(result);
			xuUnitVacuum	:= 0;
			CASE takeoverPosition OF
				1:
					product		:= xuUnit.ProductData_Get(product := 10,	clearLastProduct := FALSE, clearData := TRUE);
					statistics.Count(product);
					product		:= xuUnit.ProductData_Get(product := 7,		clearLastProduct := FALSE, clearData := TRUE);
					statistics.Count(product);
					product		:= xuUnit.ProductData_Get(product := 4,		clearLastProduct := FALSE, clearData := TRUE);
					statistics.Count(product);
					product		:= xuUnit.ProductData_Get(product := 1,		clearLastProduct := FALSE, clearData := TRUE);
					statistics.Count(product);
					PulseOutput.AddPulses(4);
					xuUnitVacuum.Vacuum01	:= TRUE;

				2:
					product		:= xuUnit.ProductData_Get(product := 11,	clearLastProduct := FALSE, clearData := TRUE);
					statistics.Count(product);
					product		:= xuUnit.ProductData_Get(product := 8,		clearLastProduct := FALSE, clearData := TRUE);
					statistics.Count(product);
					product		:= xuUnit.ProductData_Get(product := 5,		clearLastProduct := FALSE, clearData := TRUE);
					statistics.Count(product);
					product		:= xuUnit.ProductData_Get(product := 2,		clearLastProduct := FALSE, clearData := TRUE);
					statistics.Count(product);
					PulseOutput.AddPulses(4);
					xuUnitVacuum.Vacuum02	:= TRUE;

				3:
					product		:= xuUnit.ProductData_Get(product := 12,	clearLastProduct := FALSE, clearData := TRUE);
					statistics.Count(product);
					product		:= xuUnit.ProductData_Get(product := 9,		clearLastProduct := FALSE, clearData := TRUE);
					statistics.Count(product);
					product		:= xuUnit.ProductData_Get(product := 6,		clearLastProduct := FALSE, clearData := TRUE);
					statistics.Count(product);
					product		:= xuUnit.ProductData_Get(product := 3,		clearLastProduct := FALSE, clearData := TRUE);
					statistics.Count(product);
					PulseOutput.AddPulses(4);
					xuUnitVacuum.Vacuum03	:= TRUE;
			END_CASE
		END_IF

		// Xu Unit releases all vacuums; returns true after a timeout.
		result[1]	:= result[1] OR_ELSE xuUnit.ReleaseProducts(xuUnitVacuum);

		IF Timer.Set(In := Arrays.Bool_All(result, TRUE), Pt := 0.4) THEN
			ActState := StateXuUnitMovesToParking;
		END_IF

	StateXuUnitMovesToParking:
		IF State.Changed THEN
			Arrays.Bool_Reset(result);
		END_IF

		result[1]	:= result[1] OR_ELSE xuUnit.MoveToParking(almostSafe => almostSafe);

		IF Arrays.Bool_All(result, TRUE) THEN
			ActState := StateFinal;
		END_IF

	StateFinal:
		ActState := StateNone;
END_CASE
END_METHOD

// Command to stop a module (Statemachine to zero state)
METHOD PUBLIC Stop : BOOL	// Returns true when drives are in standstill
CommandLock.ForceRelease();

ActState	:= StateNone;
Stop		:= TRUE;
END_METHOD

// Transfer has started and is doing something
{attribute 'monitoring':='call'}
PROPERTY TransferBusy : BOOL
GET
VAR
END_VAR
TransferBusy	:= ActState <> StateNone;
END_GET
END_PROPERTY

(* ---- TransferProducts_XuToZFB.fb ---- *)
{attribute 'symbol' := 'none'}
{attribute 'monitoring_display' := 'ActState'}
FUNCTION_BLOCK TransferProducts_XuToZFB
EXTENDS Transfer_BaseFB
IMPLEMENTS IModuleTransferExecute
VAR_INPUT
	xuUnit					: IXuUnit_Default_Transfer_Commands;
	zUnit					: IZUnit_Transfer_Commands;
END_VAR
VAR
	result					: ARRAY[1..2] OF BOOL;

	ActState :
	(
		StateNone							:= 0,
		StateZUnitMovesInPosition			:= 100,
		StateCheckIfTransferNeeded			:= 200,
		StateXuUnitMovesToTakeover			:= 300,
		StateZUnitGetsProducts				:= 400,
		StateXuUnitReleasesProducts			:= 500,
		StateXuUnitMovesToParking			:= 600,
		StateFreeZUnit						:= 700,
		StateFinal							:= 999
	) DINT;

END_VAR

SUPER^();

// Enable manual control of Z Unit motor when Xu Unit is in safe position.
zUnit.ExternalManualControlEnabled := xuUnit.InSafePos;

END_FUNCTION_BLOCK

// Check if a transfer is needed
METHOD PUBLIC CheckIfTransferIsNeeded : BOOL
VAR_INPUT
	iParameter			: INT := 1;	// 0: Invalid, 1: Takeover Pos 1, etc.
END_VAR
// Xu unit has at least 1 product in the gripper. We need a transfer.
CheckIfTransferIsNeeded	S= xuUnit.HasPayload <> enumPayload.None;

// Running in semi-auto mode without setting vacuums.
CheckIfTransferIsNeeded	S= SER.OperationMode = SER_OperationModeType.SemiAuto AND HMI.SemiAutoMode = enumSemiAutoModeType.WithoutVacuums;

//CheckIfTransferIsNeeded	S= SER.OperationMode = SER_OperationModeType.SemiAuto AND PersistentVars.RecipeVars.ActiveExchangeSet = enumExchangeSets.FourCavDualTakeover;
END_METHOD

METHOD PROTECTED Cyclic
State(actState	:= ActState);
END_METHOD

// Command to reset the module (Statemachine to zero state) in case of E-Stop
METHOD PUBLIC EStop : BOOL	// Returns true when drives are in standstill
CommandLock.ForceRelease();

ActState	:= StateNone;
EStop		:= TRUE;
END_METHOD

// After a state change, this method is called to execute the current state
METHOD PROTECTED Execute
CASE PersistentVars.RecipeVars.ActiveExchangeSet OF
//	enumExchangeSets.SingleCavSingleTakeover:
//		Execute_Sequence1();
//	enumExchangeSets.SingleCavDualTakeover:
//		Execute_Sequence2();
//	enumExchangeSets.FourCavDualTakeover:
//		Execute_Sequence3();
//	enumExchangeSets.TwoCavSingleTakeover:
//		Execute_Sequence4();
	ELSE
		ShowNoProgramWarning();
		Execute_Sequence1();
END_CASE
END_METHOD

// Start transfer of products or labels between 2 units
METHOD PUBLIC ExecuteTransfer : BOOL
VAR_INPUT
	iParameter : INT := 1;	// 0: Invalid, 1: Takeover Pos 1, etc.
END_VAR
IF NOT CommandLock.Request(__POUNAME()) THEN
	RETURN;
END_IF

IF CommandLock.FirstCall THEN
	;
END_IF

takeoverPosition := iParameter;	// Copy parameters

IF ActState = StateNone THEN
	ActState := StateZUnitMovesInPosition;
END_IF

IF ActState = StateFinal THEN
	ExecuteTransfer := CommandLock.Release(__POUNAME());
END_IF
END_METHOD

METHOD PROTECTED Execute_Sequence1
IF State.Changed THEN
	Arrays.Bool_Reset(result);
END_IF

CASE ActState OF
	StateNone:
		;

	StateZUnitMovesInPosition:
		// Check if the z unit does not have any products on the gripper.
		IF NOT zUnit.ReadyForTransfer THEN
			RETURN;
		END_IF

		// Check if all products are present on the Xu Unit gripper.
		// Or the cycle has just started, the first cycle it is allowed to transfer an incomplete gripper.
		IF xuUnit.HasPayload = enumPayload._All
		OR SER.OperationMode = SER_OperationModeType.SemiAuto
		OR SER.ActState = PACK_ML.State.Starting
		THEN
			IF (result[1] OR_ELSE (result[1] := zUnit.MoveToTakeover(1)))
			THEN
				ActState := StateXuUnitMovesToTakeover;
			END_IF
		END_IF

	StateXuUnitMovesToTakeover:
		IF  (result[1] OR_ELSE (result[1] := xuUnit.MoveToTakeover(1)))
		THEN
			ActState := StateZUnitGetsProducts;
		END_IF

	StateZUnitGetsProducts:
		IF State.Changed THEN
			zUnit.CopyProductStatus(
				takeoverPos	:= 1,
				productNo	:= 1,
				product		:= xuUnit.ProductData_Get(product := 1));
		END_IF

		xuUnit.ReleaseProducts(AllVacuums);

		// Z Unit gets products; returns true when all vacuums are high
		IF zUnit.GetProducts(vacuumIndex := 2#0010) THEN
			ActState := StateXuUnitReleasesProducts;
		END_IF

	StateXuUnitReleasesProducts:
		// Xu Unit releases all vacuums; returns true after a timeout.
		IF xuUnit.ReleaseProducts(AllVacuums) THEN
			ActState := StateXuUnitMovesToParking;
		END_IF

	StateXuUnitMovesToParking:
		IF xuUnit.MoveToParking() THEN
			ActState := StateFreeZUnit;
		END_IF

	StateFreeZUnit:
		// The last step of the product transfer must always be: TransferComplete()
		// This lets the Z Unit know that the transfer is done.
		// The Z Unit decides if it moves to the next Takeover position, or stack the products.
		IF zUnit.TransferComplete(0) THEN
			ActState := StateFinal;
		END_IF

	StateFinal:
		ActState := StateNone;
END_CASE
END_METHOD

METHOD PROTECTED Execute_Sequence2
IF State.Changed THEN
	Arrays.Bool_Reset(result);
END_IF

CASE ActState OF
	StateNone:
		;

	StateZUnitMovesInPosition:
		// Check if the z unit does not have any products on the gripper.
		IF NOT zUnit.ReadyForTransfer THEN
			RETURN;
		END_IF

		// Check if all products are present on the Xu Unit gripper.
		// Or the cycle has just started, the first cycle it is allowed to transfer an incomplete gripper.
		IF xuUnit.HasPayload = enumPayload._All
		OR SER.OperationMode = SER_OperationModeType.SemiAuto
		OR SER.ActState = PACK_ML.State.Starting
		THEN
			IF (result[1] OR_ELSE (result[1] := zUnit.MoveToTakeover(1)))
			THEN
				ActState := StateXuUnitMovesToTakeover;
			END_IF
		END_IF

	StateXuUnitMovesToTakeover:
		IF  (result[1] OR_ELSE (result[1] := xuUnit.MoveToTakeover(1)))
		THEN
			ActState := StateZUnitGetsProducts;
		END_IF

	StateZUnitGetsProducts:
		IF State.Changed THEN
			zUnit.CopyProductStatus(
				takeoverPos	:= 1,
				productNo	:= SEL(takeoverPosition = 1, 2, 1),
				product		:= xuUnit.ProductData_Get(product := 1));
		END_IF

		xuUnit.ReleaseProducts(AllVacuums);

		// Z Unit gets products; returns true when all vacuums are high
		IF zUnit.GetProducts(vacuumIndex := SEL(takeoverPosition = 1, 2#0100, 2#0010)) THEN
			ActState := StateXuUnitReleasesProducts;
		END_IF

	StateXuUnitReleasesProducts:
		// Xu Unit releases all vacuums; returns true after a timeout.
		IF xuUnit.ReleaseProducts(AllVacuums) THEN
			ActState := StateXuUnitMovesToParking;
		END_IF

	StateXuUnitMovesToParking:
		IF xuUnit.MoveToParking() THEN
			ActState := StateFreeZUnit;
		END_IF

	StateFreeZUnit:
		// The last step of the product transfer must always be: TransferComplete()
		// This lets the Z Unit know that the transfer is done.
		// The Z Unit decides if it moves to the next Takeover position, or stack the products.
		IF zUnit.TransferComplete(takeoverPosition) THEN

			// If all products are transferred to the gripper, reset the counter to 1.
			IF NOT zUnit.ReadyForTransfer THEN
				AlternateCycleCounter := 1;
			ELSE
				AlternateCycleCounter := AlternateCycleCounter + 1;
			END_IF

			ActState := StateFinal;
		END_IF

	StateFinal:
		ActState := StateNone;
END_CASE
END_METHOD

METHOD PROTECTED Execute_Sequence3
IF State.Changed THEN
	Arrays.Bool_Reset(result);
END_IF

CASE ActState OF
	StateNone:
		;

	StateZUnitMovesInPosition:
		// Check if the z unit does not have any products on the gripper.
		IF NOT zUnit.ReadyForTransfer THEN
			RETURN;
		END_IF

		// Check if all products are present on the Xu Unit gripper.
		// Or the cycle has just started, the first cycle it is allowed to transfer an incomplete gripper.
		IF xuUnit.HasPayload = enumPayload._All
		OR (xuUnit.HasPayload = enumPayload._Any AND takeoverPosition = 2)
		OR SER.OperationMode = SER_OperationModeType.SemiAuto
		OR SER.ActState = PACK_ML.State.Starting
		THEN
			IF (result[1] OR_ELSE (result[1] := zUnit.MoveToTakeover(takeoverPosition)))
			THEN
				ActState := StateXuUnitMovesToTakeover;
			END_IF
		END_IF

	StateXuUnitMovesToTakeover:
		IF  (result[1] OR_ELSE (result[1] := xuUnit.MoveToTakeover(1)))
		THEN
			ActState := StateZUnitGetsProducts;
		END_IF

	StateZUnitGetsProducts:
		IF State.Changed THEN
			zUnit.CopyProductStatus(
				takeoverPos	:= takeoverPosition,
				productNo	:= 1,
				product		:= xuUnit.ProductData_Get(product := SEL(takeoverPosition = 1, 3, 1), clearData := TRUE));
			zUnit.CopyProductStatus(
				takeoverPos	:= takeoverPosition,
				productNo	:= 2,
				product		:= xuUnit.ProductData_Get(product := SEL(takeoverPosition = 1, 4, 2), clearData := TRUE));
		END_IF

		xuUnit.ReleaseProducts(SEL(takeoverPosition = 1, 2#0100, 2#0010));

		// Z Unit gets products; returns true when all vacuums are high
		IF zUnit.GetProducts(vacuumIndex := SEL(takeoverPosition = 1, 2#0100, 2#0010)) THEN
			ActState := StateXuUnitReleasesProducts;
		END_IF

	StateXuUnitReleasesProducts:
		// Xu Unit releases all vacuums; returns true after a timeout.
		IF xuUnit.ReleaseProducts(SEL(takeoverPosition = 1, 2#0100, 2#0010)) THEN
			ActState := StateXuUnitMovesToParking;
		END_IF

	StateXuUnitMovesToParking:
		IF takeoverPosition = 1 THEN
			xuUnit.MoveToHalfway();
			ActState := StateFreeZUnit;
		ELSIF xuUnit.MoveToParking() THEN
			ActState := StateFreeZUnit;
		END_IF

	StateFreeZUnit:
		IF zUnit.TransferComplete(takeoverPosition) THEN
			ActState := StateFinal;
		END_IF

	StateFinal:
		ActState := StateNone;
END_CASE
END_METHOD

METHOD PROTECTED Execute_Sequence4
IF State.Changed THEN
	Arrays.Bool_Reset(result);
END_IF

CASE ActState OF
	StateNone:
		;

	StateZUnitMovesInPosition:
		// Check if the z unit does not have any products on the gripper.
		IF NOT zUnit.ReadyForTransfer THEN
			RETURN;
		END_IF

		// Check if all products are present on the Xu Unit gripper.
		// Or the cycle has just started, the first cycle it is allowed to transfer an incomplete gripper.
		IF xuUnit.HasPayload = enumPayload._All
		OR SER.OperationMode = SER_OperationModeType.SemiAuto
		OR SER.ActState = PACK_ML.State.Starting
		THEN
			IF (result[1] OR_ELSE (result[1] := zUnit.MoveToTakeover(1)))
			THEN
				ActState := StateXuUnitMovesToTakeover;
			END_IF
		END_IF

	StateXuUnitMovesToTakeover:
		IF  (result[1] OR_ELSE (result[1] := xuUnit.MoveToTakeover(1)))
		THEN
			ActState := StateZUnitGetsProducts;
		END_IF

	StateZUnitGetsProducts:
		IF State.Changed THEN
			zUnit.CopyProductStatus(
				takeoverPos	:= 1,
				productNo	:= 1,
				product		:= xuUnit.ProductData_Get(product := 1));
			zUnit.CopyProductStatus(
				takeoverPos	:= 1,
				productNo	:= 2,
				product		:= xuUnit.ProductData_Get(product := 2));
		END_IF

		xuUnit.ReleaseProducts(AllVacuums);

		// Z Unit gets products; returns true when all vacuums are high
		IF zUnit.GetProducts(vacuumIndex := 2#0110) THEN
			ActState := StateXuUnitReleasesProducts;
		END_IF

	StateXuUnitReleasesProducts:
		// Xu Unit releases all vacuums; returns true after a timeout.
		IF xuUnit.ReleaseProducts(AllVacuums) THEN
			ActState := StateXuUnitMovesToParking;
		END_IF

	StateXuUnitMovesToParking:
		IF xuUnit.MoveToParking() THEN
			ActState := StateFreeZUnit;
		END_IF

	StateFreeZUnit:
		// The last step of the product transfer must always be: TransferComplete()
		// This lets the Z Unit know that the transfer is done.
		// The Z Unit decides if it moves to the next Takeover position, or stack the products.
		IF zUnit.TransferComplete(0) THEN
			ActState := StateFinal;
		END_IF

	StateFinal:
		ActState := StateNone;
END_CASE
END_METHOD

// Command to stop a module (Statemachine to zero state)
METHOD PUBLIC Stop : BOOL	// Returns true when drives are in standstill
CommandLock.ForceRelease();

ActState	:= StateNone;
Stop		:= TRUE;
END_METHOD

// Transfer has started and is doing something
{attribute 'monitoring':='call'}
PROPERTY TransferBusy : BOOL
GET
VAR
END_VAR
TransferBusy	:= ActState <> StateNone;
END_GET
END_PROPERTY
